{attribute addProperty BoxType "EL5151-0021-0018"}
{attribute addProperty Id "ENC_StatusAT %I*ENC_Status_053BC81D80100ENC_Filtered_latchAT %I*ENC_Filtered_latch_7F6716946480ENC_ControlAT %Q*ENC_Control_E047A95D112140WcStateAT %I*WcState_98A4DF7520.250InfoDataAT %I*InfoData_BC63D37F80100"}
{attribute addProperty CRC "3008258255"}
{attribute addProperty SizeInBites "338"}
{attribute addProperty SizeInBytes "42.25"}
TYPE EL5151_0683EF8C :
STRUCT
	{attribute addProperty Name "ENC_Status"}
	ENC_Status : ENC_Status_053BC81D;
	{attribute addProperty Name "ENC_Filtered_latch"}
	ENC_Filtered_latch : ENC_Filtered_latch_7F671694;
	{attribute addProperty Name "ENC_Control"}
	ENC_Control : ENC_Control_E047A95D;
	{attribute addProperty Name "WcState"}
	WcState : WcState_98A4DF75;
	{attribute addProperty Name "InfoData"}
	InfoData : InfoData_BC63D37F;
END_STRUCT
END_TYPE

(* stored: Version 1.2.0.0, ProductVersion 3.1.4024.9
   DUT EL5151_0683EF8C: Id {b22022cc-b401-4bac-b67c-d82c9d80053d} *)
